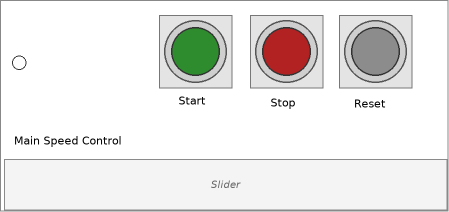
VISUALIZATION Visu2_MainCtr  // 449x212
    Slider (4,159 443x51), variable: stIO.stIn.iSetSpeedMotor, scale 0..100
    RadioButton (10,14 150x97), variable: stParam.stStatus.eMMA
        Areas[0]: Text=Mode Init
        Areas[1]: Text=Mode Auto
        Areas[2]: Text=Mode Manual
    PushSwitch (159,15 73x73), tooltip "Start", variable: stIO.stIn.xStartIO, behaviour: TAP, style: Switch-PushSwitch-Green
    PushSwitch (250,15 73x73), tooltip "Stop", variable: stIO.stIn.xStopIO, invisible if: fbMMA.iEtape<>350, behaviour: TAP, style: Switch-PushSwitch-Red
    PushSwitch (339,15 73x73), tooltip "Reset", variable: stIO.stIn.xResetIO, behaviour: TAP, style: Switch-PushSwitch-Gray
    Label (152,86 80x30), "Start"
    Label (243,88 80x30), "Stop", invisible if: fbMMA.iEtape<>350
    Label (330,89 80x30), "Reset", invisible if: fbMMA.iEtape<>350
    Label (11,126 176x30), "Main Speed Control"
END_VISUALIZATION

(* stored: Version 1.1.0.1, ProductVersion 3.1.4020.12
   Visu Visu2_MainCtr: Id {f89229b0-9fbe-4658-9615-7efd65a8d1ae} *)
